// TwinCAT 3 PLC project ourPLC
// ProgramVersion: 3.1.4026.20
// CompilerDefines: VISU_USEPROPERTYINFO
// libraries:
//   CmpBitmapPool, * (System)
//   Tc2_Standard, * (Beckhoff Automation GmbH)
//   Tc2_System, * (Beckhoff Automation GmbH)
//   VisuDialogs, * (System)
// project tree:
//   DUTs/ trafficlight_cmds_typ.TcDUT, trafficLight_counters_typ.TcDUT, trafficLight_inputs_typ.TcDUT (not stored), trafficLight_outputs_typ.TcDUT, trafficLight_state_enum.TcDUT, trafficlight_state_typ.TcDUT, trafficLight_timers_typ.TcDUT (not stored), trafficlight_transitions_typ.TcDUT, trafficLight_typ.TcDUT
//   / GlobalTextList.TcGTLO, ImagePool.TcIPO (not stored), PlcTask.TcTTO, Visualization Manager.TcVMO (not stored), VISU_TASK.TcTTO
//   POUs/ MAIN.TcPOU (not stored), outHandler.TcPOU (not stored), transitionLogic.TcPOU (not stored)
//   VISUs/ mainPage.TcVIS, disconnected.TcVIS
// real-time tasks:
//   TASK PlcTask: cycle T#10ms, priority 20, ADS port 350
//   TASK VISU_TASK: cycle T#200000us, priority 30, ADS port 351
// I/O:
//   DEVICE Device 2 (EtherCAT), AmsNetId 5.144.153.185.3.1
//     Term 1 (EK1100) [EK1100 EtherCAT Coupler (2A E-Bus)]
//       Term 2 (EL5101) [EL5101 1Ch. Inc. Encoder 5V]
//       Term 3 (EL2008) [EL2008 8Ch. Dig. Output 24V, 0.5A]
//       Term 4 (EL4031) [EL4031 1Ch. Ana. Output +/-10V, 12bit]
//       Term 5 (EL1008) [EL1008 8Ch. Dig. Input 24V, 3ms]
//       Term 6 (EL9011) [EL9011 End Terminal]
// variable links:
//   ourPLC/ourPLC Instance <-> Device 2 (EtherCAT)/Term 1 (EK1100)/Term 3 (EL2008)
//     PlcTask Outputs/MAIN.mytrafficlight.outputs.GREENlight <-> Channel 5/Output
//     PlcTask Outputs/MAIN.mytrafficlight.outputs.REDlight <-> Channel 1/Output
//     PlcTask Outputs/MAIN.mytrafficlight.outputs.YELLOWlight <-> Channel 3/Output
//   ourPLC/ourPLC Instance <-> Device 2 (EtherCAT)/Term 1 (EK1100)/Term 5 (EL1008)
//     PlcTask Inputs/MAIN.capacitive <-> Channel 2/Input
//     PlcTask Inputs/MAIN.mytrafficlight.inputs.iGreenINPUT <-> Channel 5/Input
//     PlcTask Inputs/MAIN.mytrafficlight.inputs.iRedINPUT <-> Channel 7/Input
//     PlcTask Inputs/MAIN.mytrafficlight.inputs.iSwitchOffINPUT <-> Channel 1/Input
//     PlcTask Inputs/MAIN.mytrafficlight.inputs.iSwitchOnINPUT <-> Channel 3/Input

CONFIGURATION ourPLC
    RESOURCE PLC ON TwinCAT3
        TASK PlcTask(INTERVAL := T#10ms, PRIORITY := 20);
        TASK VISU_TASK(INTERVAL := T#200000us, PRIORITY := 30);
        PROGRAM MAIN WITH PlcTask : MAIN;
        PROGRAM VisuElems_Visu_Prg WITH VISU_TASK : VisuElems.Visu_Prg;
    END_RESOURCE
END_CONFIGURATION

// ---- DUTs/trafficlight_cmds_typ.TcDUT
TYPE trafficlight_cmds_typ :
STRUCT
	cmdStart:BOOL;
END_STRUCT
END_TYPE

// ---- DUTs/trafficLight_counters_typ.TcDUT
TYPE trafficLight_counters_typ :
STRUCT
	timerGreen   : TON; // Timer para la luz verde
    timerYellow   : TON; // Timer para la luz ámbar
    timerRed    : TON; // Timer para la luz roja
	timerBlink :TON;
	timerconfig1 : TON;
	timerconfig2 : TON;
	timerconfig3 : TON;
END_STRUCT
END_TYPE

// ---- DUTs/trafficLight_outputs_typ.TcDUT
TYPE trafficLight_outputs_typ :
STRUCT
	REDlight AT %Q*: BOOL;
	GREENlight AT %Q*: BOOL;
	YELLOWlight AT %Q*: BOOL;
END_STRUCT
END_TYPE

// ---- DUTs/trafficLight_state_enum.TcDUT
{attribute 'qualified_only'}
{attribute 'strict'}
TYPE trafficLight_state_enum :
(
	A1_DISCONNECTED := 0,
	F1_stYELLOW := 1,
	F1_stRED := 2,
	F1_stGREEN := 3,
	F2_stBLINKon := 4,
	F2_stBLINKoff := 5,
	F6_stYELLOW := 6,
	F6_stRED :=7,
	F6_stGREEN :=8
);
END_TYPE

// ---- DUTs/trafficlight_state_typ.TcDUT
TYPE trafficlight_state_typ :
STRUCT
	state: trafficLight_state_enum := trafficLight_state_enum.A1_DISCONNECTED;
	state_str: STRING := 'stDisabled';
END_STRUCT
END_TYPE

// ---- DUTs/trafficlight_transitions_typ.TcDUT
TYPE trafficlight_transitions_typ :
STRUCT
	power_on_Done :BOOL;
	yellow_Done: BOOL;
	green_Done: BOOL;
	red_Done:BOOL;
	blinkON_Done: BOOL;
	blinkOFF_Done: BOOL;
	power_down_ack: BOOL;
	
END_STRUCT
END_TYPE

// ---- DUTs/trafficLight_typ.TcDUT
TYPE trafficLight_typ :
STRUCT
	
	state: trafficLight_state_typ;
	timers: trafficLight_timers_typ;
	counters: trafficLight_counters_typ;
	outputs: trafficLight_outputs_typ;
	cmds:trafficLight_cmds_typ;
	transitions: trafficLight_transitions_typ;
	inputs: trafficLight_inputs_typ;
	
	
END_STRUCT
END_TYPE

// ---- GlobalTextList.TcGTLO
TEXTLIST GlobalTextList
  382 = '%s'
  130 = 'CAT'
  152 = 'CATALÀ'
  282 = 'CATALÁ'
  69 = 'DESCONECTADO'
  404 = 'DISCONNECT'
  671 = 'EL HMI DEL SEMÁFORO'
  872 = 'ENG'
  287 = 'ENGLSH'
  876 = 'ESP'
  258 = 'EUS'
  518 = 'EUSKERA'
  208 = 'OFF'
  512 = 'ON/OFF'
  364 = 'TRAFFIC LIGHT HMI' | EUSKERA: 'SEMAFOROAREN HMIa' | CATALÀ: "L'HMI DEL SEMÀFOR" | ENGLISH: 'THE TRAFFIC LIGHT HMI'
  INST_OFF = 'Sistema apagado.\nActive el interruptor para iniciar.' | EUSKERA: 'Sistema itzalita.\nPiztu etengailua hasteko.' | CATALÀ: "Sistema apagat.\nActivi l'interruptor per iniciar." | ENGLISH: 'System off.\nTurn on the switch to start.'
  INST_WAIT = 'Modo Espera (Parpadeo).\nPulse BOTÓN VERDE para inicio.' | EUSKERA: 'Itxarote modua (Keinuka).\nSakatu BOTOI BERDEA hasteko.' | CATALÀ: 'Mode espera (Parpelleig).\nPremi BOTÓ VERD per iniciar.' | ENGLISH: 'Standby mode (Blinking).\nPress GREEN BUTTON to start.'
  INST_NORMAL = 'Funcionamiento Normal.\nPulse BOTÓN ROJO para Setup.' | EUSKERA: 'Funtzionamendu normala.\nSakatu BOTOI GORRIA konfiguratzeko.' | CATALÀ: 'Funcionament normal.\nPremi BOTÓ VERMELL per al Setup.' | ENGLISH: 'Normal operation.\nPress RED BUTTON for Setup.'
  INST_SETUP_Y = 'Setup: Tiempo AMARILLO.\nPulse BOTÓN ROJO para guardar.' | EUSKERA: 'Setup: Horiaren denbora.\nSakatu BOTOI GORRIA gordetzeko.' | CATALÀ: 'Setup: Temps GROC.\nPremi BOTÓ VERMELL per guardar.' | ENGLISH: 'Setup: YELLOW time.\nPress RED BUTTON to save.'
  INST_SETUP_R = 'Setup: Tiempo ROJO.\nPulse BOTÓN ROJO para guardar.' | EUSKERA: 'Setup: Gorriaren denbora.\nSakatu BOTOI GORRIA gordetzeko.' | CATALÀ: 'Setup: Temps VERMELL.\nPremi BOTÓ VERMELL per guardar.' | ENGLISH: 'Setup: RED time.\nPress RED BUTTON to save.'
  INST_SETUP_G = 'Setup: Tiempo VERDE.\nPulse BOTÓN ROJO para terminar.' | EUSKERA: 'Setup: Berdearen denbora.\nSakatu BOTOI GORRIA amaitzeko.' | CATALÀ: 'Setup: Temps VERD.\nPremi BOTÓ VERMELL per acabar.' | ENGLISH: 'Setup: GREEN time.\nPress RED BUTTON to finish.'
END_TEXTLIST

// ---- VISUs/mainPage.TcVIS
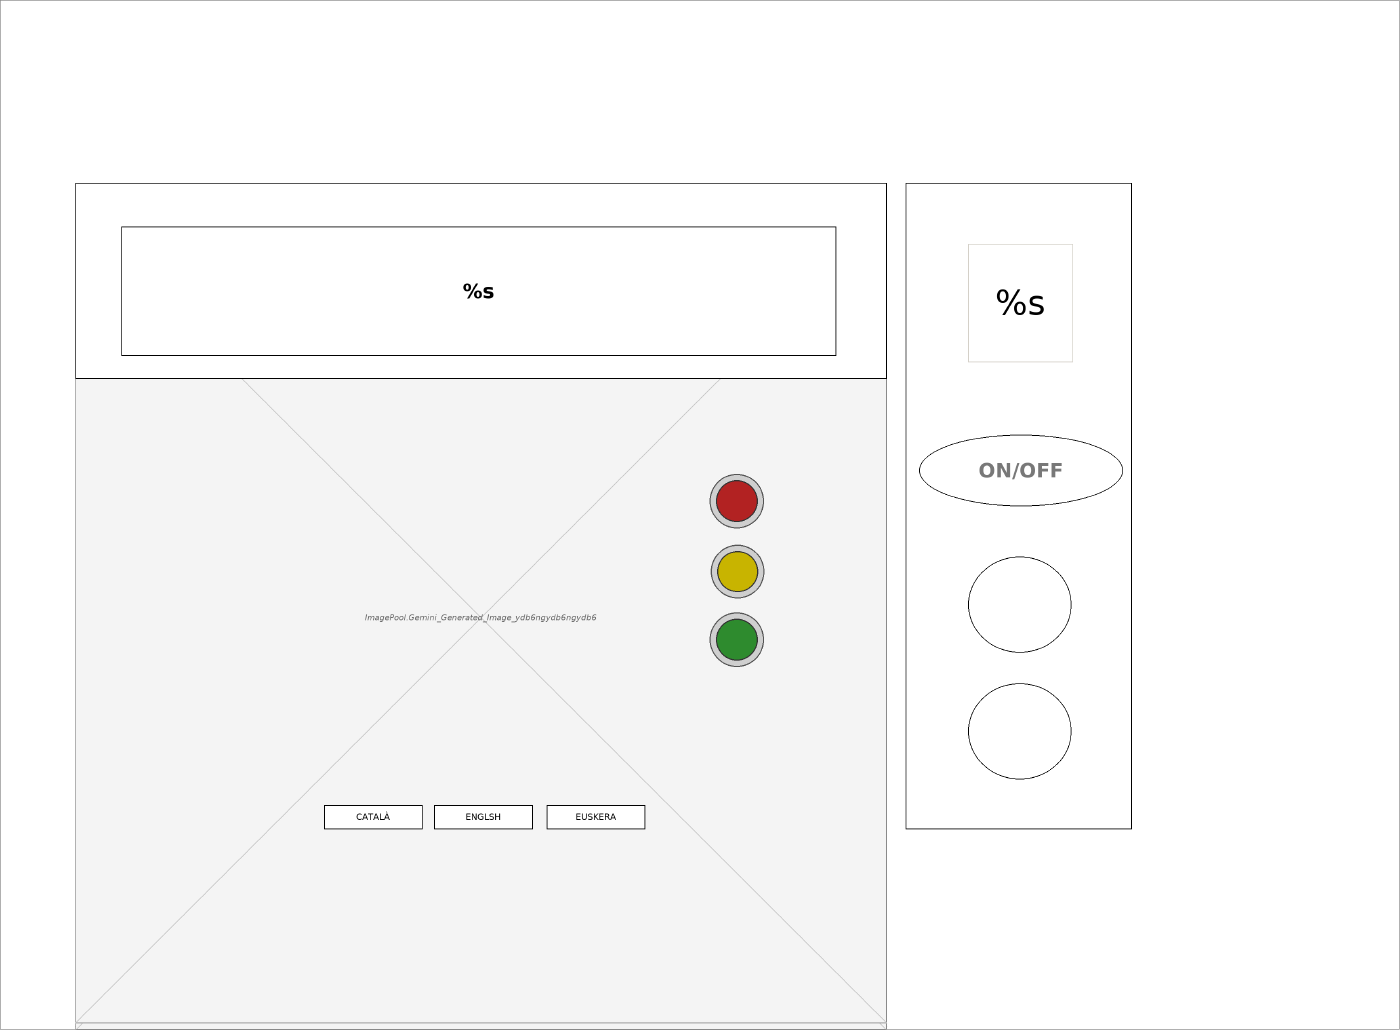
VISUALIZATION mainPage  // 1767x1301
    Image (95,272 1024x1024), invisible if: MAIN.boolENG, image: ImagePool.1772114357870
    RoundedRectangle (951,388 816x285), angle 90
    Image (95,253 1024x1048), invisible if: MAIN.boolCAT, image: ImagePool.Gemini_Generated_Image_6byr8p6byr8p6byr - copia
    Image (95,268 1024x1024), invisible if: MAIN.boolEUS, image: ImagePool.Gemini_Generated_Image_ydb6ngydb6ngydb6
    RoundedRectangle (95,231 1024x247)
    Lamp1 (890,593 80x80), variable: MAIN.mytrafficlight.outputs.REDlight, style: Lamp-Lamp1-Red
    Lamp1 (891,683 80x78), variable: MAIN.mytrafficlight.outputs.YELLOWlight, style: Lamp-Lamp1-Yellow
    Lamp1 (890,768 80x80), variable: MAIN.mytrafficlight.outputs.GREENlight, style: Lamp-Lamp1-Green
    Label (424,246 395x30), "EL HMI DEL SEMÁFORO"
    Ellipse (1222,703 130x121), colour toggle: MAIN.mytrafficlight.inputs.iGreen
        tap MAIN.mytrafficlight.inputs.iGreen
    Ellipse (1222,863 130x121), colour toggle: MAIN.mytrafficlight.inputs.iRed
        tap MAIN.mytrafficlight.inputs.iRed p1329445385=TRUE
    Ellipse (1160,549 257x90), "ON/OFF"
        toggle MAIN.updateState.HMI_Switch
    RoundedRectangle (409,1017 124x30), "CATALÀ"
        toggle MAIN.boolCAT
        OnMouseClick: ChangeLanguage ChangeLanguage=CATALÀ
        OnMouseClick: execute {
            MAIN.boolCAT := FALSE;
            MAIN.boolENG := TRUE;
            MAIN.boolEUS := TRUE;
        }
    RoundedRectangle (548,1017 124x30), "ENGLSH"
        OnMouseClick: ChangeLanguage ChangeLanguage=ENGLISH
        OnMouseClick: execute {
            MAIN.boolCAT := TRUE;
            MAIN.boolEUS := TRUE;
            MAIN.boolENG := FALSE;
        }
    RoundedRectangle (690,1017 124x30), "EUSKERA"
        toggle MAIN.boolEUS
        OnMouseClick: ChangeLanguage ChangeLanguage=EUSKERA
        OnMouseClick: execute {
            MAIN.boolCAT := TRUE;
            MAIN.boolENG := TRUE;
            MAIN.boolEUS := FALSE;
        }
    Textfield (1222,308 132x149), "%s", text variable: MAIN.visuTIME
        p4168582468: MAIN.visuTIME
    Rectangle (153,286 902x163), "%s", text list: 'GlobalTextList', text index: MAIN.mensajeIdioma
END_VISUALIZATION

// ---- VISUs/disconnected.TcVIS
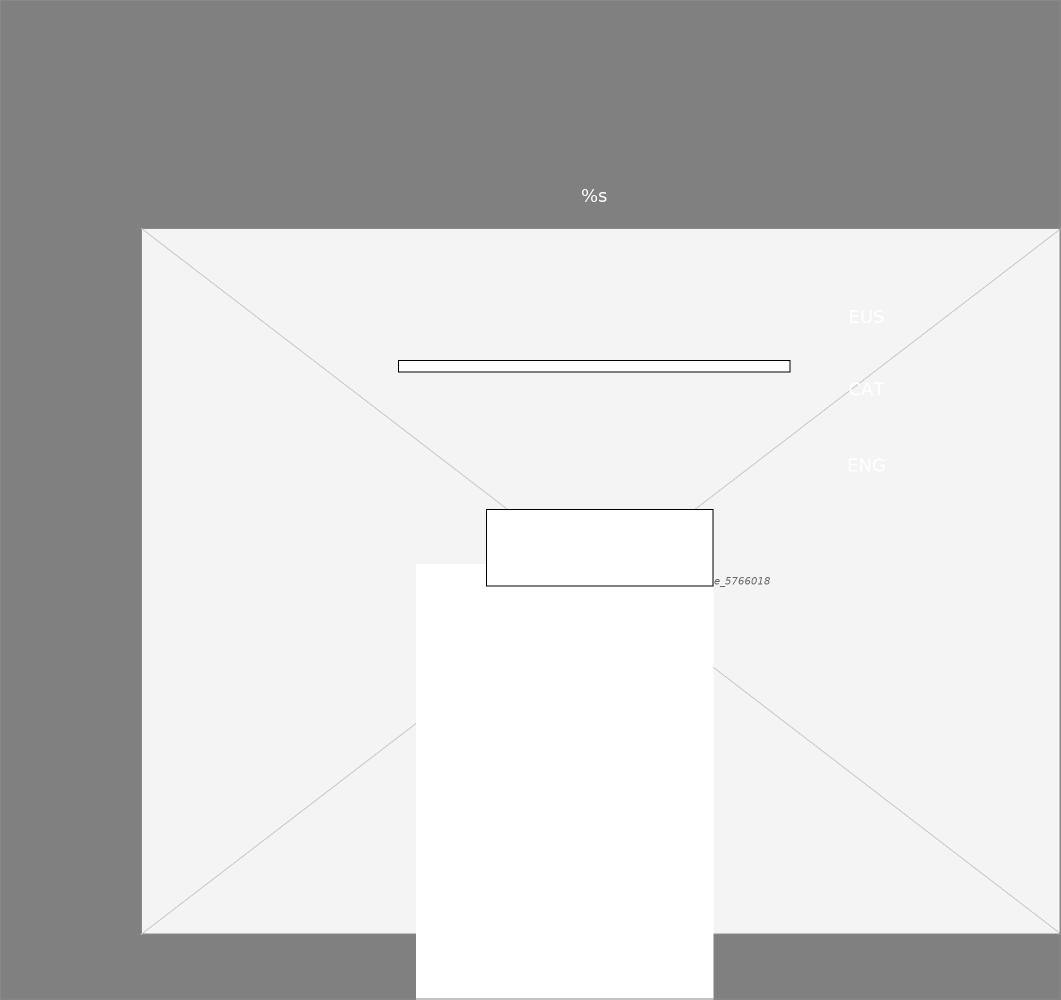
VISUALIZATION disconnected  // 1061x1000
    Image (141,228 920x706), image: ImagePool.pngtree-traffic-lights-clipart-design-png-image_5766018
    Rectangle (398,360 392x12), angle 315
    Rectangle (416,564 297x436)
    RoundedRectangle (486,509 227x77), "ON/OFF"
        toggle MAIN.updateState.HMI_Switch
        OnMouseClick: change screen: mainPage
    RoundedRectangle (424,161 341x70), "%s", text list: 'GlobalTextList', text index: MAIN.mensajeIdioma
    Rectangle (754,287 225x60), "EUS"
        OnMouseClick: ChangeLanguage ChangeLanguage=EUSKERA
        OnMouseClick: execute {
            main.boolCAT := TRUE;
            main.boolENG := TRUE;
            main.boolEUS := FALSE;
        }
    Rectangle (754,357 225x65), "CAT"
        OnMouseClick: ChangeLanguage ChangeLanguage=CATALÀ
        OnMouseClick: execute {
            main.boolCAT := FALSE;
            main.boolENG := TRUE;
            main.boolEUS := TRUE;
        }
    Rectangle (754,436 225x59), "ENG"
        OnMouseClick: ChangeLanguage ChangeLanguage=ENGLISH
        OnMouseClick: execute {
            main.boolCAT := TRUE;
            main.boolENG := FALSE;
            main.boolEUS := TRUE;
        }
END_VISUALIZATION
